TEXTLIST TL_AuswahlSchrauberAblauf
  0 = 'Reset Ablauf'
  1 = 'Original Ablauf'
  2 = 'Entwickelung Ablauf'
   = ''
END_TEXTLIST

(* stored: Version 1.1.0.1, ProductVersion 3.1.4024.15
   TextList TL_AuswahlSchrauberAblauf: Id {7965f445-936b-4ade-95ed-2915821e3927} *)
